TYPE TcoUrRoboticsT2OFloatRegs :
STRUCT
    {attribute addProperty Name "<#Float registers#>"}
    Register : ARRAY[0..23] OF REAL;
END_STRUCT
END_TYPE

(* stored: Version 1.1.0.1, ProductVersion 3.1.4024.12
   DUT TcoUrRoboticsT2OFloatRegs: Id {bf5a76cf-ab69-003f-1aa4-d04b0642bc88} *)
